PROGRAM P_Outputs
VAR
	fbWinchValveOutput 		: FB_ValveOutput;
	fbCylValveOutput 		: FB_ValveOutput;
END_VAR

///////////////////// Winch //////////////////////////////
G_Outputs.stWinchValveOutput.bEnable := G_Work.bManualMode OR G_Work.bAutoMode; 

fbWinchValveOutput(
	bEnable := G_Work.bWinchEnable OR G_Work.fWinchTime > 0.0,
	bDeadBandCompOn := G_Parameters.stParam.bDeadBandCompOn,
	stValveDeadBand := G_Parameters.stParam.stWinchValveDeadBand,
	fNormalizedInput := G_Work.fWinchControlInput,
	nOutput => G_Outputs.stWinchValveOutput.nValveOutput
);

///////////////////// Cylinder //////////////////////////////
G_Outputs.stCylValveOutput.bEnable := G_Work.bManualMode OR G_Work.bAutoMode;

fbCylValveOutput(
	bEnable := G_Work.bCylEnable OR G_Work.fCylTime > 0.0,
	bDeadBandCompOn := G_Parameters.stParam.bDeadBandCompOn,
	stValveDeadBand := G_Parameters.stParam.stCylValveDeadBand,
	fNormalizedInput := G_Work.fCylControlInput,
	nOutput => G_Outputs.stCylValveOutput.nValveOutput
);

END_PROGRAM

(* stored: Version 1.1.0.1, ProductVersion 3.1.4024.11
   POU P_Outputs: Id {05725e2c-789e-4faf-9ddc-3f7ec72a2093}, SpecialFunc None *)
